{attribute 'linkalways'} 
{attribute 'no_explicit_call' := 'This FB is a CLASS and must be accessed using methods or properties'}
{attribute 'enable_dynamic_creation'}
FUNCTION_BLOCK Node_F_VN_ApplyTranslationToAffineTransformation EXTENDS VisionNode
VAR
    aTransformationMatrix : _TcVnMatrix2x3_LREAL;
    fDeltaX : _LREAL(0.0);
    fDeltaY : _LREAL(0.0);
    hrPrev : _HRESULT(S_OK);
	hresult : _HRESULT(S_OK);
END_VAR

METHOD PUBLIC  Clone : I_Node
VAR
	pNode : POINTER TO Node_F_VN_ApplyTranslationToAffineTransformation;
END_VAR
pNode := __NEW(Node_F_VN_ApplyTranslationToAffineTransformation);
Clone := pNode^;
END_METHOD

METHOD FB_init : BOOL
VAR_INPUT
	bInitRetains : BOOL; // if TRUE, the retain variables are initialized (warm start / cold start)
	bInCopyCode : BOOL;  // if TRUE, the instance afterwards gets moved into the copy code (online change)
END_VAR
AddInput('aTransformationMatrix', aTransformationMatrix);
AddParameter('fDeltaX', fDeltaX);
AddParameter('fDeltaY', fDeltaY);
AddInput('hrPrev', hrPrev);
AddOutput('aTransformationMatrix', aTransformationMatrix);
AddOutput('hresult',hresult);
END_METHOD

METHOD PROTECTED  OnExecute : HRESULT
hresult.Value := F_VN_ApplyTranslationToAffineTransformation(
	aTransformationMatrix := aTransformationMatrix.Value,
    fDeltaX := fDeltaX.Value,
    fDeltaY := fDeltaY.Value,
	hrPrev := hrPrev.Value);
END_METHOD

METHOD PUBLIC PreExecutionCheck
VAR_INPUT
	Check : I_PreExecutionChecks;
END_VAR
END_METHOD

END_FUNCTION_BLOCK

(* stored: Version 1.1.0.1, ProductVersion 3.1.4024.13
   POU Node_F_VN_ApplyTranslationToAffineTransformation: Id {0b1c03cf-edeb-0ef1-1dbb-810d55efff7b}, SpecialFunc None
   Folder Constructor: Id {77f9fc11-f623-048d-2bcc-3d706aded1fa}
   Method Clone: Id {0ccf611a-3165-05c5-1854-44080aeb2447}
   Method FB_init: Id {1589010f-d1fd-0f6f-17fe-741f543edda7}
   Method OnExecute: Id {760c6e73-56a4-03e5-265c-e6e4f8b341d7}
   Method PreExecutionCheck: Id {08b7934a-5159-0f64-2487-7e31f5990a9d} *)
